TYPE ST_ProfidriveCuConfig :
STRUCT
	stRecordIdent		: ST_RecordIdent;
END_STRUCT
END_TYPE

(* stored: Version 1.1.0.1, ProductVersion 3.1.4024.12
   DUT ST_ProfidriveCuConfig: Id {b31645a5-bde5-01b1-2946-142992e72a60} *)
